// TIA Portal project "Counter Sayıcılar Uygulama" (V17)

(* hardware
DEVICE "S71500/ET200MP-Station_1"  S7-1500 station
   slot 0: "Profilschiene_0"  6ES7 590-1***0-0AA0
   slot 1: "PLC_1"  CPU 1511-1 PN  6ES7 511-1AK00-0AB0  V1.8
   slot 2: "AI 8xU/I/RTD/TC ST_1"  AI 8xU/I/RTD/TC ST  6ES7 531-7KF00-0AB0  V2.0
   slot 3: "AI 8xU/I/RTD/TC ST_2"  AI 8xU/I/RTD/TC ST  6ES7 531-7KF00-0AB0  V2.0
   slot 4: "AI 8xU/I/RTD/TC ST_3"  AI 8xU/I/RTD/TC ST  6ES7 531-7KF00-0AB0  V2.0
   slot 5: "AI 8xU/I/RTD/TC ST_4"  AI 8xU/I/RTD/TC ST  6ES7 531-7KF00-0AB0  V2.0
   slot 6: "DI 16x24VDC BA_1"  DI 16x24VDC BA  6ES7 521-1BH10-0AA0  V1.0
*)

// ===== PLC "PLC_1"  CPU 1511-1 PN =====

VAR_GLOBAL   // PLC tag table "Standard-Variablentabelle"
   "START" AT %E0.0 : Bool;
   "1.KONVEYOR" AT %A0.0 : Bool;
   "1.SENSOR" AT %E0.1 : Bool;
   "Tag_1" AT %M0.0 : Bool;
   "2.SENSOR" AT %I0.2 : Bool;
   "Tag_2" AT %M10.0 : Bool;
   "2.KONVEYOR" AT %Q0.1 : Bool;
   "3.SENSOR" AT %I0.3 : Bool;
   "3.KONVEYOR" AT %Q0.2 : Bool;
   "Tag_3" AT %M0.1 : Bool;
   "Tag_4" AT %M10.1 : Bool;
   "Tag_5" AT %M10.2 : Bool;
END_VAR

// folder: System blocks/Program resources

DATA_BLOCK "IEC_Counter_0_DB"   // DB1
{ S7_Optimized_Access := 'TRUE' }
AUTHOR : Simatic
FAMILY : IEC
NAME : CNTR
VERSION : 1.0
// stored: InstanceOfName IEC_COUNTER
"IEC_COUNTER"
BEGIN
END_DATA_BLOCK

// folder: (top level)

FUNCTION "MHJ-PLC-Lab-Function-S71500" : Void   // FC9000, SCL
{ S7_Optimized_Access := 'TRUE' }
VERSION : 0.1
   VAR_TEMP
      Value : Byte;
      ForCounter : Int;
   END_VAR
   VAR CONSTANT
      Value_01_DW : DWord := 16#1223_5486;
      Value_02_DW : DWord := 16#A6C9_D1F5;
   END_VAR
BEGIN

   #Value:=PEEK(area := 16#82,
        dbNumber := 0,
        byteOffset := 511);
   #Value := #Value + 1;

   POKE(area := 16#82,
        dbNumber := 0,
        byteOffset := 511,
        value := #Value);

   POKE(area := 16#82,
        dbNumber := 0,
        byteOffset := 1016,
        value := #Value_01_DW);
   POKE(area := 16#82,
        dbNumber := 0,
        byteOffset := 1020,
        value := #Value_02_DW);

   FOR #ForCounter := 0 TO 63 DO
       #Value:=PEEK(area := 16#1,
            dbNumber := 0,
            byteOffset := #ForCounter);
       POKE(area := 16#81,
            dbNumber := 0,
            byteOffset := #ForCounter,
            value := #Value);
   END_FOR;
   #Value := PEEK(area := 16#1,
                  dbNumber := 0,
                  byteOffset := 512);
   POKE(area := 16#82,
        dbNumber := 0,
        byteOffset := 512,
        value := #Value);
END_FUNCTION

ORGANIZATION_BLOCK "Main"   // OB1, LAD, ProgramCycle
TITLE = "Main Program Sweep (Cycle)"
{ S7_Optimized_Access := 'TRUE' }
VERSION : 0.1
   VAR_INPUT
      Initial_Call : Bool;   // Initial call of this OB
      Remanence : Bool;   // =True, if remanent data are available
   END_VAR
   VAR_TEMP   // added for the SCL form of the ladder/FBD networks
      _w1 : Bool;
   END_VAR
BEGIN

REGION Network 1
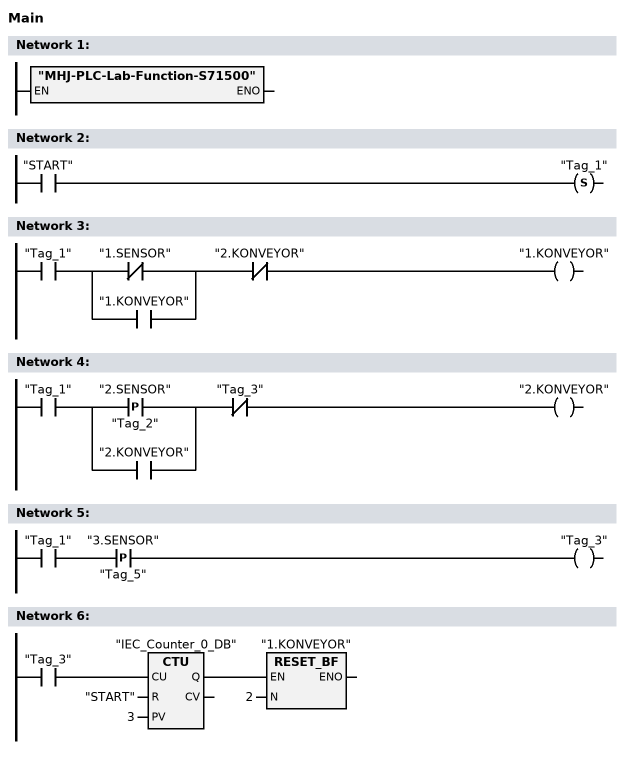
   RUNG wire#powerrail
      "MHJ-PLC-Lab-Function-S71500"()
   END_RUNG
   // the same network as SCL:
   "MHJ-PLC-Lab-Function-S71500"();
END_REGION

REGION Network 2
   RUNG wire#powerrail
      Contact( "START" )
      S_Coil( "Tag_1" )
   END_RUNG
   // the same network as SCL:
   IF "START" THEN "Tag_1" := TRUE; END_IF;
END_REGION

REGION Network 3
   RUNG wire#powerrail
      Contact( "Tag_1" )
      wire#w1
      I_Contact( "1.SENSOR" )
      wire#w2
      I_Contact( "2.KONVEYOR" )
      Coil( "1.KONVEYOR" )
   END_RUNG
   RUNG wire#w1
      Contact( "1.KONVEYOR" )
   END_RUNG wire#w2
   // the same network as SCL:
   "1.KONVEYOR" := "Tag_1" AND (NOT "1.SENSOR" OR "1.KONVEYOR") AND NOT "2.KONVEYOR";
END_REGION

REGION Network 4
   RUNG wire#powerrail
      Contact( "Tag_1" )
      wire#w1
      P_Contact(operand := "2.SENSOR", bit := "Tag_2")
      wire#w2
      I_Contact( "Tag_3" )
      Coil( "2.KONVEYOR" )
   END_RUNG
   RUNG wire#w1
      Contact( "2.KONVEYOR" )
   END_RUNG wire#w2
   // the same network as SCL:
   #_w1 := "Tag_1" AND "2.SENSOR" AND NOT "Tag_2";   // rising edge of "2.SENSOR"
   "Tag_2" := "2.SENSOR";
   "2.KONVEYOR" := (#_w1 OR ("Tag_1" AND "2.KONVEYOR")) AND NOT "Tag_3";
END_REGION

REGION Network 5
   RUNG wire#powerrail
      Contact( "Tag_1" )
      P_Contact(operand := "3.SENSOR", bit := "Tag_5")
      Coil( "Tag_3" )
   END_RUNG
   // the same network as SCL:
   #_w1 := "Tag_1" AND "3.SENSOR" AND NOT "Tag_5";   // rising edge of "3.SENSOR"
   "Tag_5" := "3.SENSOR";
   "Tag_3" := #_w1;
END_REGION

REGION Network 6
   // no SCL statement known for RBitfield: written as a call
   "IEC_Counter_0_DB".CTU(CU := "Tag_3", R := "START", PV := 3);
   IF "IEC_Counter_0_DB".Q THEN RESET_BF(operand := "1.KONVEYOR", n := 2); END_IF;
END_REGION
END_ORGANIZATION_BLOCK